{attribute 'qualified_only'}
{attribute 'strict'}
TYPE E_Sensor :
(
	Sick := 0,
	Pilz := 1,
	Parker := 2,
	Bosch := 3
);
END_TYPE

(* stored: Version 1.1.0.1, ProductVersion 3.1.4024.12
   DUT E_Sensor: Id {1ed943b1-c9bd-4275-80be-7c6cb397c36f} *)
